SUBAPPLICATION Uebung_072c (* GBSD auf UT ausgeben *)
  (* Standard: 61499-2; Description: Copyright (c) 2023 Meisterschulen am Ostbahnhof This program and the accompanying materials are made available under the terms of the Eclipse Public License 2.0 which is available at https://www.eclipse.org/legal/epl-2.0/ SPDX-License-Identifier: EPL-2.0 *)
  (* Version 1.0, 2023-10-23, Franz Höpfinger, Meisterschulen am Ostbahnhof *)
  PACKAGE Uebungen;
  IMPORT Uebungen::const::UT::DefaultPool_TECU::NumberVariable_Ground_based_machine_speed;
  IMPORT Uebungen::const::UT::DefaultPool_TECU::NumberVariable_Wheel_based_machine_distance;
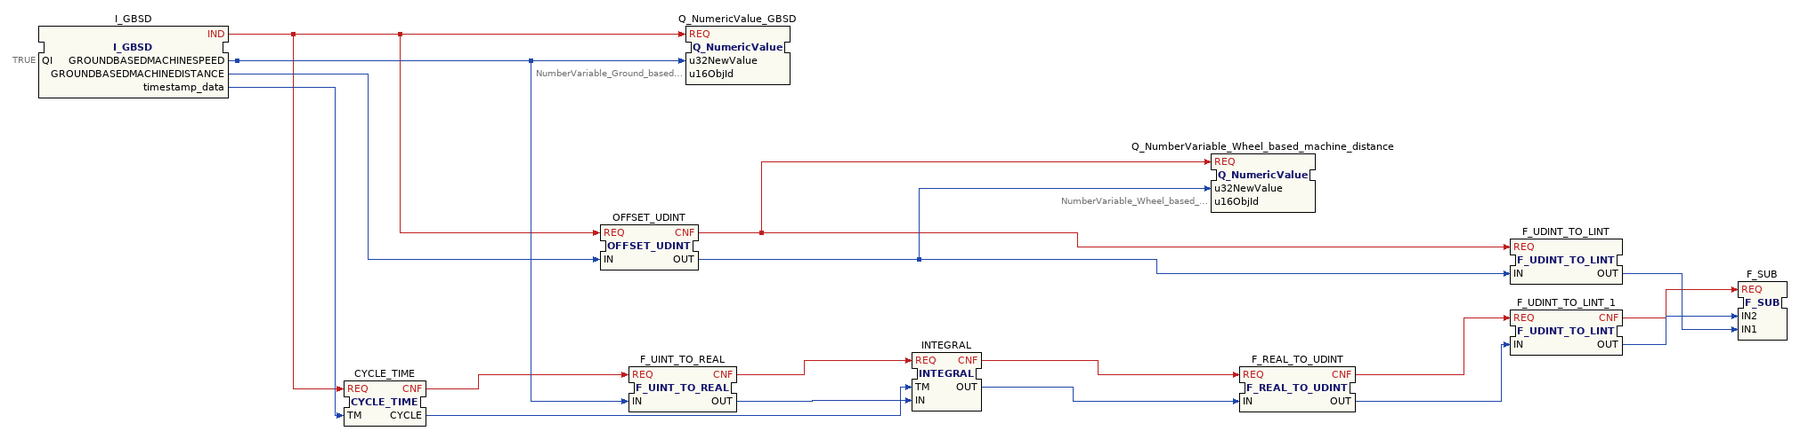
  FBS
    I_GBSD : isobus::tecu::I_GBSD(QI := TRUE);
    Q_NumericValue_GBSD : isobus::ut::Q_NumericValue(u16ObjId := NumberVariable_Ground_based_machine_speed);
    Q_NumberVariable_Wheel_based_machine_distance : isobus::ut::Q_NumericValue(u16ObjId := NumberVariable_Wheel_based_machine_distance);
    INTEGRAL : logiBUS::utils::math::INTEGRAL;
    OFFSET_UDINT : logiBUS::utils::math::OFFSET_UDINT;
    CYCLE_TIME : utils::timing::CYCLE_TIME;
    F_UINT_TO_REAL : iec61131::conversion::F_UINT_TO_REAL;
    F_REAL_TO_UDINT : iec61131::conversion::F_REAL_TO_UDINT;
    F_SUB : iec61131::arithmetic::F_SUB;
    F_UDINT_TO_LINT : iec61131::conversion::F_UDINT_TO_LINT;
    F_UDINT_TO_LINT_1 : iec61131::conversion::F_UDINT_TO_LINT;
  END_FBS
  EVENT_CONNECTIONS
    I_GBSD.IND TO Q_NumericValue_GBSD.REQ;
    I_GBSD.IND TO OFFSET_UDINT.REQ;
    OFFSET_UDINT.CNF TO Q_NumberVariable_Wheel_based_machine_distance.REQ;
    I_GBSD.IND TO CYCLE_TIME.REQ;
    CYCLE_TIME.CNF TO F_UINT_TO_REAL.REQ;
    F_UINT_TO_REAL.CNF TO INTEGRAL.REQ;
    INTEGRAL.CNF TO F_REAL_TO_UDINT.REQ;
    F_REAL_TO_UDINT.CNF TO F_UDINT_TO_LINT_1.REQ;
    OFFSET_UDINT.CNF TO F_UDINT_TO_LINT.REQ;
    F_UDINT_TO_LINT_1.CNF TO F_SUB.REQ;
  END_CONNECTIONS
  DATA_CONNECTIONS
    I_GBSD.GROUNDBASEDMACHINESPEED TO Q_NumericValue_GBSD.u32NewValue;
    I_GBSD.GROUNDBASEDMACHINEDISTANCE TO OFFSET_UDINT.IN;
    OFFSET_UDINT.OUT TO Q_NumberVariable_Wheel_based_machine_distance.u32NewValue;
    I_GBSD.timestamp_data TO CYCLE_TIME.TM;
    CYCLE_TIME.CYCLE TO INTEGRAL.TM;
    F_UINT_TO_REAL.OUT TO INTEGRAL.IN;
    I_GBSD.GROUNDBASEDMACHINESPEED TO F_UINT_TO_REAL.IN;
    INTEGRAL.OUT TO F_REAL_TO_UDINT.IN;
    OFFSET_UDINT.OUT TO F_UDINT_TO_LINT.IN;
    F_REAL_TO_UDINT.OUT TO F_UDINT_TO_LINT_1.IN;
    F_UDINT_TO_LINT_1.OUT TO F_SUB.IN2;
    F_UDINT_TO_LINT.OUT TO F_SUB.IN1;
  END_CONNECTIONS
END_SUBAPPLICATION
